FUNCTION_BLOCK FB_TransportLogik
VAR_INPUT
	eStateE : eBetriebszustand;
	bEnable : BOOL;
	bExecute : BOOL;
	nStation : INT;
	
	bStation1 : BOOL;
	bStation2 : BOOL;
	bStation3 : BOOL;
	bStation4 : BOOL;
END_VAR
VAR_OUTPUT
	eStateA : eBetriebszustand;
	bEnableA : BOOL;
	bExecuteA : BOOL;
	bHaltA : BOOL;
	
	bStop1 : BOOL;
	bStop2 : BOOL;
	bStop3 : BOOL;
END_VAR
VAR
	nState : INT;
END_VAR

CASE nState OF
	0: //OFF
	eStateA := eBetriebszustand.OFF;
	
	bEnableA := FALSE;
	bExecuteA := FALSE;
	bHaltA := FALSE;
	bStop1 := FALSE;
	bStop2 := FALSE;
	bStop3 := FALSE;
	
	IF bEnable THEN
		nState := 1;
	END_IF
	
	1: //INIT
	eStateA := eBetriebszustand.INIT;
	
	bEnableA := TRUE;
	bExecuteA := FALSE;
	bHaltA := FALSE;
	bStop1 := FALSE;
	bStop2 := FALSE;
	bStop3 := FALSE;
	
	IF eStateE = eBetriebszustand.READY THEN
		nState := 2;
	END_IF
	
	2: //READY
	eStateA := eBetriebszustand.READY;
	
	bEnableA := TRUE;
	bExecuteA := FALSE;
	bHaltA := TRUE;
	bStop1 := FALSE;
	bStop2 := FALSE;
	bStop3 := FALSE;
	
	IF bExecute THEN
		nState := 3;
	END_IF
	
	3: //PROD-Förderband start
	eStateA := eBetriebszustand.PROD;
	
	bEnableA := TRUE;
	bExecuteA := TRUE;
	bHaltA := FALSE;
	IF (nStation - 1) = 1 THEN
		bStop1 := TRUE;
		bStop2 := FALSE;
		bStop3 := FALSE;
	ELSIF (nStation - 1) = 2 THEN
		bStop1 := FALSE;
		bStop2 := TRUE;
		bStop3 := FALSE;
	ELSIF (nStation - 1) = 3 THEN
		bStop1 := FALSE;
		bStop2 := FALSE;
		bStop3 := TRUE;
	END_IF
	
	IF bStation1 AND nStation = 1 THEN
		nState := 4;
	ELSIF bStation2 AND nStation = 2 THEN
		nState := 4;
	ELSIF bStation3 AND nStation = 3 THEN
		nState := 4;
	ELSIF bStation4 AND nStation = 4 THEN
		nState := 4;
	END_IF
	
	4: //PROD-Förderband stop
	eStateA := eBetriebszustand.PROD;
	
	bEnableA := TRUE;
	bExecuteA := FALSE;
	bHaltA := TRUE;
	bStop1 := FALSE;
	bStop2 := FALSE;
	bStop3 := FALSE;
	
	IF eStateE = eBetriebszustand.READY THEN
		nState := 5;
	END_IF
	
	5: //DONE
	eStateA := eBetriebszustand.DONE;
	
	IF NOT bExecute THEN
		nState := 2;
	END_IF
END_CASE

END_FUNCTION_BLOCK

(* stored: Version 1.1.0.1, ProductVersion 3.1.4024.15
   POU FB_TransportLogik: Id {e1b20b99-cc52-4075-8608-92d62d8ecdb3}, SpecialFunc None *)
